{attribute 'linkalways'} 
{attribute 'no_explicit_call' := 'This FB is a CLASS and must be accessed using methods or properties'}
{attribute 'enable_dynamic_creation'}
FUNCTION_BLOCK EventHandlerItemOnceOnly EXTENDS EventHandlerItem
VAR
	parent : I_EventEmitter;
END_VAR

METHOD PUBLIC Emit
VAR_INPUT
	EventName : T_MaxString;
	Event : I_Event;
END_VAR
SUPER^.Emit(EventName,Event);
parent.OffEvent(name,handler);
END_METHOD

METHOD FB_init : BOOL
VAR_INPUT
	bInitRetains : BOOL; // if TRUE, the retain variables are initialized (warm start / cold start)
	bInCopyCode : BOOL;  // if TRUE, the instance afterwards gets moved into the copy code (online change)
	Name : T_MAXSTRING;
	Handler : I_EventHandler;
	Parent : I_EventEmitter;
END_VAR
THIS^.parent := Parent;
END_METHOD

END_FUNCTION_BLOCK

(* stored: Version 1.1.0.1, ProductVersion 3.1.4024.12
   POU EventHandlerItemOnceOnly: Id {fe48e8b4-7ae4-4438-9da4-8ee2563092e3}, SpecialFunc None
   Folder Constructor: Id {842a482e-a238-4285-af46-d80720fa60ac}
   Method Emit: Id {17f8c72e-1b12-4a24-bf07-283947ac7690}
   Method FB_init: Id {81d52a11-588d-4036-aaac-a9abca8bf4fe} *)
